FUNCTION_BLOCK IXA (* Composite FB for boolean input data *)
  (* Standard: 61499-2; Description: Copyright (c) 2024 HR Agrartechnik GmbH This program and the accompanying materials are made available under the terms of the Eclipse Public License 2.0 which is available at https://www.eclipse.org/legal/epl-2.0/ SPDX-License-Identifier: EPL-2.0 *)
  (* Version 1.0, 2024-04-24, franz *)
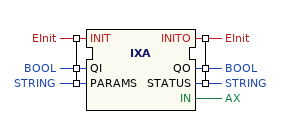
  EVENT_INPUT
    INIT : EInit WITH QI, PARAMS; (* Service Initialization *)
  END_EVENT
  EVENT_OUTPUT
    INITO : EInit WITH QO, STATUS; (* Initialization Confirm *)
  END_EVENT
  VAR_INPUT
    QI : BOOL; (* Event Input Qualifier *)
    PARAMS : STRING; (* Service Parameters *)
  END_VAR
  VAR_OUTPUT
    QO : BOOL; (* Event Output Qualifier *)
    STATUS : STRING; (* Service Status *)
  END_VAR
  PLUGS
    IN : AX;
  END_PLUGS
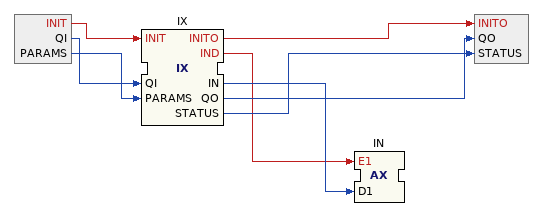
  FBS
    IX : IX;
  END_FBS
  EVENT_CONNECTIONS
    INIT TO IX.INIT;
    IX.INITO TO INITO;
    IX.IND TO IN.E1;
  END_CONNECTIONS
  DATA_CONNECTIONS
    IX.IN TO IN.D1;
    QI TO IX.QI;
    PARAMS TO IX.PARAMS;
    IX.QO TO QO;
    IX.STATUS TO STATUS;
  END_CONNECTIONS
END_FUNCTION_BLOCK
